Staubli VAL3: TrajItem.pjx

--- TrajItem.pjx ---
Parameters version=s7.5 stackSize=5000 millimeterUnit=true
Data file=TrajItem.dtx
Type name=TrajectoryItem path=Disk://kernel/template/TrajectoryItem/TrajectoryItem.pjx

--- TrajItem.dtx ---
public TrajectoryItem tSuper
  [0]
    num distance
    num moveType
    num nTime
    num nStop
    num nTcpAction
    string comment
    bool toStop
    mdesc nom_speed = {vel=450, tmax=1000}
    InstrItem iInstr[3]
      [0]
        string sType
        string sData
      [1]
        string sType
        string sData
      [2]
        string sType
        string sData
    num nMoveId
public pointRx pPoint
public num nType
public pointRx pCircle
